TYPE DUT_SKILL_INPUT :
STRUCT
	///Range of parameters
	ParameterInput: ARRAY[0..ParameterCnt] OF DUT_PARAMETER_INPUT;
	///Start process
	Execute: BOOL;
END_STRUCT
END_TYPE

(* stored: Version 1.1.0.1, ProductVersion 3.1.0.25
   DUT DUT_SKILL_INPUT: Id {ae665477-9417-4c9d-88c7-665baf638eb1} *)
